{attribute 'GeneratedUsingTerminal: EL2521-1001-0000'}
{attribute addProperty BoxType "EL2521-1001-0000"}
{attribute addProperty Id "InputsAT %I*Inputs_0292EF133OutputsAT %Q*Outputs_905E7D863WcStateAT %I*WcState_9091E0EB2InfoDataAT %I*InfoData_32EB74EA10"}
{attribute addProperty CRC "1429073621"}
{attribute addProperty Size "18"}
TYPE EL2521_552DEED5 EXTENDS EtcSlaveTerminalBase_947E5A46 :
STRUCT
	{attribute addProperty Name "Inputs"}
	Inputs : Inputs_0292EF13;
	{attribute addProperty Name "Outputs"}
	Outputs : Outputs_905E7D86;
	{attribute addProperty Name "WcState"}
	WcState : WcState_9091E0EB;
	{attribute addProperty Name "InfoData"}
	InfoData : InfoData_32EB74EA;
END_STRUCT
END_TYPE

(* stored: Version 1.2.0.0, ProductVersion 3.1.4024.9
   DUT EL2521_552DEED5: Id {1e5bbd7d-f56f-44d6-ab06-796e342acec1} *)
